PROGRAM P_Motion
VAR

END_VAR

P_FastScan();
P_Z_Axis();
P_SlowScan();

END_PROGRAM

(* stored: Version 1.1.0.1, ProductVersion 3.1.4024.11
   POU P_Motion: Id {a07fa915-69b4-42b1-8b6d-ccc4cf561082}, SpecialFunc None *)
